(*~
<docu>
	<summary>
		`TcoAi` status structure.								
	</summary>				
</docu>	
~*)
TYPE
    TcaLaserDistanceSenorStatus :
    STRUCT
		{attribute addProperty Name "<#Raw range#>"}
        RawRange : REAL;
		{attribute addProperty Name "<#Real range#>"}
        RealRange : REAL;
		{attribute addProperty Name "<#Scaled value#>"}
        Scaled : REAL;
    END_STRUCT
END_TYPE

(* stored: Version 1.1.0.1
   DUT TcaLaserDistanceSenorStatus: Id {0321329e-083a-4947-a873-ff9645cee8a8} *)
